{attribute 'GeneratedUsingTerminal: EK1960-2600-0021'}
{attribute addProperty BoxType "EK1960-2600-0021"}
{attribute addProperty Id "FSoE_InputsFSoE_Inputs_A1F422BE48FSoE_OutputsFSoE_Outputs_37DEC56456"}
{attribute addProperty CRC "3079329168"}
{attribute addProperty Size "104"}
TYPE Module_1_FSoE_B78AD590 :
STRUCT
	{attribute addProperty Name "FSoE_Inputs"}
	FSoE_Inputs  : FSoE_Inputs_A1F422BE;
	{attribute addProperty Name "FSoE_Outputs"}
	FSoE_Outputs  : FSoE_Outputs_37DEC564;
END_STRUCT
END_TYPE

(* stored: Version 1.2.0.0, ProductVersion 3.1.4024.9
   DUT Module_1_FSoE_B78AD590: Id {0264f1d8-d1ec-4aa1-ba29-815f07d4a9df} *)
